RoboDK station: cinta con rodillos.rdk

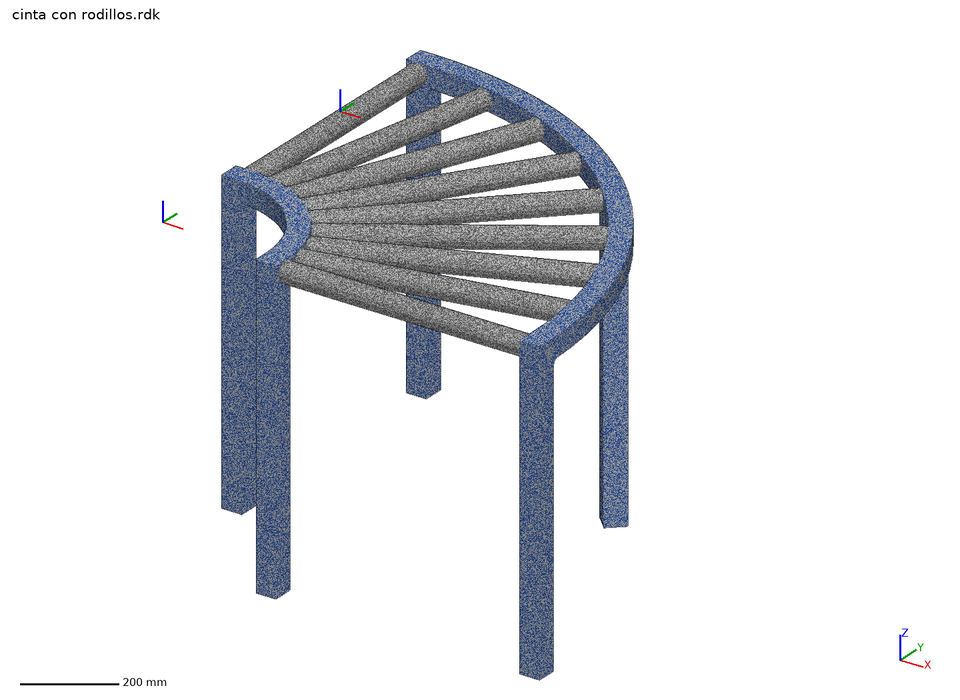
[picture v0: the station drawn from its stored meshes, robots at their saved joint values, targets as dots, program paths as lines]
Station cinta con rodillos (saved by RoboDK 5.7.4). Poses are relative to the parent item; angles as X-Y-Z fixed-axis rotations.
  - object Curva v6 at (0, 0, 0) mm, size 980 x 980 x 750 mm, geometry from Curva v6.step
  - frame Mi Mecanismo Base at (0, 0, 750) mm
    - robot Mi Mecanismo: 1 axes
        modified DH rows (alpha deg, a mm, theta deg, d mm): 0, 0, 0, 0
        joint limits [-90] to [0]; home [0]; saved at [0]
      - frame Frame 1 at (0, 625, 0) mm
